// TIA Portal V16 export
// export: Created 2022-07-21T09:35:18.9169309Z, ExportSetting WithDefaults, DisplayName Totally Integrated Automation Portal, DisplayVersion V16 Update 4, DisplayName TIA Portal Version Control Interface, DisplayVersion V16 Update 2, DisplayName TIA Portal Openness, DisplayVersion V16 Update 4, DisplayName SINAMICS Startdrive Advanced, DisplayVersion V16 Update 5, DisplayName SINAMICS Startdrive G130, G150, S120, S150, SINAMICS MV, S210, DisplayVersion V16 Update 5, DisplayName SINAMICS Startdrive G110M, G120, G120C, G120D, G120P, G115D, DisplayVersion V16 Update 5, DisplayName STEP 7 Professional, DisplayVersion V16 Update 4, DisplayName STEP 7 Safety, DisplayVersion V16, DisplayName WinCC Advanced, DisplayVersion V16 Update 4
FUNCTION_BLOCK "fbVersaStandardCom"   // FB22, LAD
TITLE = Blok do komunikacji z Versa
{ S7_Optimized_Access := 'TRUE' }
VERSION : 0.1
// stored: AutoNumber true, IsIECCheckEnabled false, IsRetainMemResEnabled false, MemoryReserve 100, SetENOAutomatically false, UDAEnableTagReadback false
   VAR_INPUT
      hwAdr : HW_IO;   // Hardware ID modułu
      dataFromSafety : Bool;
      heaterOn : Bool;   // Załączenie grzałek (=1)
      motorsOn : Bool;   // Wszystkie silniki włącz (=1)
      pump1On : Bool;   // Udostępnienie silnika 1 ON (=1)
      pump2On : Bool;   // Udostępnienie silnika 2 ON (=1)
      standbyOn : Bool;   // Załącz czuwanie (=1)
      autoOn : Bool;   // Tryb automatyczny (=1)
      maxRpm : Int := 80;   // Maksymalna predkość pomp wg. nastaw Nordson
   END_VAR
   VAR_OUTPUT
      dataSendError : Bool;   // Bład podczas wysyłki TG
      dataReceiveError : Bool;   // Błąd podczas pobierania TG
      incorrectParam : Bool;   // Niepoprawne parametry do Nordsona
      SpeedLine1Perc : Int;   // Predkość linii po konwersji prędkości pompy
      SpeedLine2Perc : Int;   // Predkość linii po konwersji prędkości pompy
   END_VAR
   VAR_IN_OUT
      monitoringError : "typeNordsonMonitoring";
      device : "typeNordson";
   END_VAR
   VAR DB_SPECIFIC
      dataSend : "typeNordsonTGOut";
      dataReceive : "typeNordsonTGIn";
      hwAddress : HW_IO;
      retValRead : Int;
      retValSend : Int;
   END_VAR
   VAR_TEMP
      tpump1Speed : Int;   // Prędkość pompy 1
      tpump2Speed : Int;   // Prędkość pompy 2
      tFactor : Real;
      tpump1SpeedPerc : Int;   // Prędkość pompy 1
      tpump2SpeedPerc : Int;   // Prędkość pompy 2
      tMaxRpm : Real;
   END_VAR
   VAR_TEMP   // added for the SCL form of the ladder/FBD networks
      _w1 : Bool;
      _w2 : Bool;
   END_VAR
BEGIN

REGION Network 1: Załaduj adres modułu
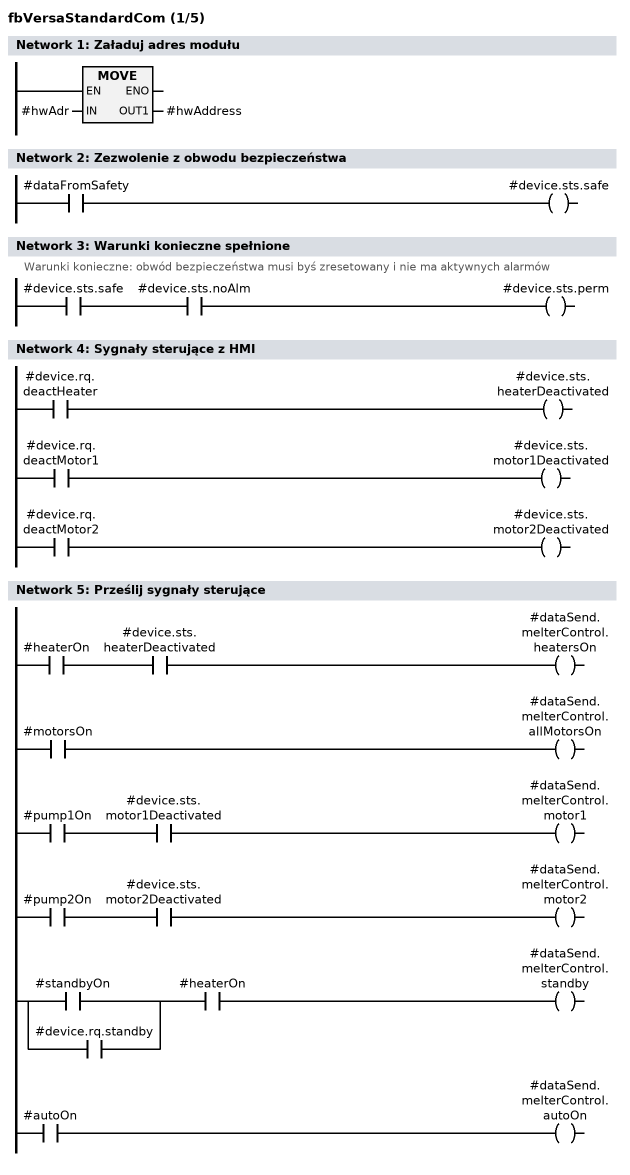
   RUNG wire#powerrail
      Move(in := #hwAdr, out1 => #hwAddress)
   END_RUNG
   // the same network as SCL:
   #hwAddress := #hwAdr;
END_REGION

REGION Network 2: Zezwolenie z obwodu bezpieczeństwa
   RUNG wire#powerrail
      Contact( #dataFromSafety )
      Coil( #device.sts.safe )
   END_RUNG
   // the same network as SCL:
   #device.sts.safe := #dataFromSafety;
END_REGION

REGION Network 3: Warunki konieczne spełnione
   // Warunki konieczne: obwód bezpieczeństwa musi byś zresetowany i nie ma aktywnych alarmów
   RUNG wire#powerrail
      Contact( #device.sts.safe )
      Contact( #device.sts.noAlm )
      Coil( #device.sts.perm )
   END_RUNG
   // the same network as SCL:
   #device.sts.perm := #device.sts.safe AND #device.sts.noAlm;
END_REGION

REGION Network 4: Sygnały sterujące z HMI
   RUNG wire#powerrail
      Contact( #device.rq.deactHeater )
      Coil( #device.sts.heaterDeactivated )
   END_RUNG
   RUNG wire#powerrail
      Contact( #device.rq.deactMotor1 )
      Coil( #device.sts.motor1Deactivated )
   END_RUNG
   RUNG wire#powerrail
      Contact( #device.rq.deactMotor2 )
      Coil( #device.sts.motor2Deactivated )
   END_RUNG
   // the same network as SCL:
   #device.sts.heaterDeactivated := #device.rq.deactHeater;
   #device.sts.motor1Deactivated := #device.rq.deactMotor1;
   #device.sts.motor2Deactivated := #device.rq.deactMotor2;
END_REGION

REGION Network 5: Prześlij sygnały sterujące
   RUNG wire#powerrail
      Contact( #heaterOn )
      Contact( #device.sts.heaterDeactivated )
      Coil( #dataSend.melterControl.heatersOn )
   END_RUNG
   RUNG wire#powerrail
      Contact( #motorsOn )
      Coil( #dataSend.melterControl.allMotorsOn )
   END_RUNG
   RUNG wire#powerrail
      Contact( #pump1On )
      Contact( #device.sts.motor1Deactivated )
      Coil( #dataSend.melterControl.motor1 )
   END_RUNG
   RUNG wire#powerrail
      Contact( #pump2On )
      Contact( #device.sts.motor2Deactivated )
      Coil( #dataSend.melterControl.motor2 )
   END_RUNG
   RUNG wire#powerrail
      Contact( #standbyOn )
      wire#w1
      Contact( #heaterOn )
      Coil( #dataSend.melterControl.standby )
   END_RUNG
   RUNG wire#powerrail
      Contact( #device.rq.standby )
   END_RUNG wire#w1
   RUNG wire#powerrail
      Contact( #autoOn )
      Coil( #dataSend.melterControl.autoOn )
   END_RUNG
   // the same network as SCL:
   #dataSend.melterControl.heatersOn := #heaterOn AND #device.sts.heaterDeactivated;
   #dataSend.melterControl.allMotorsOn := #motorsOn;
   #dataSend.melterControl.motor1 := #pump1On AND #device.sts.motor1Deactivated;
   #dataSend.melterControl.motor2 := #pump2On AND #device.sts.motor2Deactivated;
   #dataSend.melterControl.standby := (#standbyOn OR #device.rq.standby) AND #heaterOn;
   #dataSend.melterControl.autoOn := #autoOn;
END_REGION

REGION Network 6: Sprawdzanie maksymalnej prędkości 1
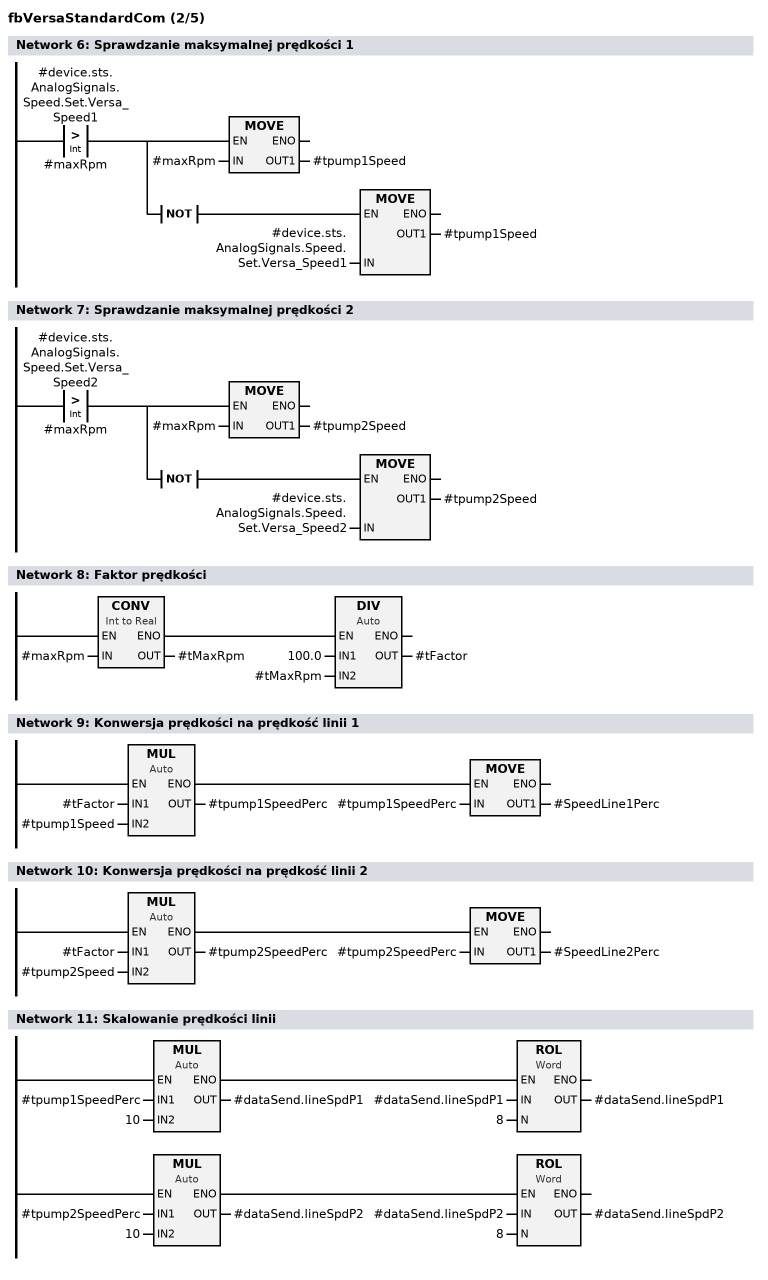
   RUNG wire#powerrail
      { S7_Templates := "SrcType := Int" } GT_Contact(in1 := #device.sts.AnalogSignals.Speed.Set.Versa_Speed1, in2 := #maxRpm)
      wire#w1
      Move(in := #maxRpm, out1 => #tpump1Speed)
   END_RUNG
   RUNG wire#w1
      Not()
      Move(in := #device.sts.AnalogSignals.Speed.Set.Versa_Speed1, out1 => #tpump1Speed)
   END_RUNG
   // the same network as SCL:
   #_w1 := #device.sts.AnalogSignals.Speed.Set.Versa_Speed1 > #maxRpm;
   IF #_w1 THEN #tpump1Speed := #maxRpm; END_IF;
   IF NOT #_w1 THEN #tpump1Speed := #device.sts.AnalogSignals.Speed.Set.Versa_Speed1; END_IF;
END_REGION

REGION Network 7: Sprawdzanie maksymalnej prędkości 2
   RUNG wire#powerrail
      { S7_Templates := "SrcType := Int" } GT_Contact(in1 := #device.sts.AnalogSignals.Speed.Set.Versa_Speed2, in2 := #maxRpm)
      wire#w1
      Move(in := #maxRpm, out1 => #tpump2Speed)
   END_RUNG
   RUNG wire#w1
      Not()
      Move(in := #device.sts.AnalogSignals.Speed.Set.Versa_Speed2, out1 => #tpump2Speed)
   END_RUNG
   // the same network as SCL:
   #_w1 := #device.sts.AnalogSignals.Speed.Set.Versa_Speed2 > #maxRpm;
   IF #_w1 THEN #tpump2Speed := #maxRpm; END_IF;
   IF NOT #_w1 THEN #tpump2Speed := #device.sts.AnalogSignals.Speed.Set.Versa_Speed2; END_IF;
END_REGION

REGION Network 8: Faktor prędkości
   RUNG wire#powerrail
      { S7_Templates := "[SrcType := Int, DestType := Real]" } Convert(in := #maxRpm, out => #tMaxRpm)
      Div(in1 := 100.0, in2 := #tMaxRpm, out => #tFactor)
   END_RUNG
   // the same network as SCL:
   #tMaxRpm := INT_TO_REAL(#maxRpm);
   #tFactor := 100.0 / #tMaxRpm;
END_REGION

REGION Network 9: Konwersja prędkości na prędkość linii 1
   RUNG wire#powerrail
      Mul(in1 := #tFactor, in2 := #tpump1Speed, out => #tpump1SpeedPerc)
      Move(in := #tpump1SpeedPerc, out1 => #SpeedLine1Perc)
   END_RUNG
   // the same network as SCL:
   #tpump1SpeedPerc := #tFactor * #tpump1Speed;
   #SpeedLine1Perc := #tpump1SpeedPerc;
END_REGION

REGION Network 10: Konwersja prędkości na prędkość linii 2
   RUNG wire#powerrail
      Mul(in1 := #tFactor, in2 := #tpump2Speed, out => #tpump2SpeedPerc)
      Move(in := #tpump2SpeedPerc, out1 => #SpeedLine2Perc)
   END_RUNG
   // the same network as SCL:
   #tpump2SpeedPerc := #tFactor * #tpump2Speed;
   #SpeedLine2Perc := #tpump2SpeedPerc;
END_REGION

REGION Network 11: Skalowanie prędkości linii
   #dataSend.lineSpdP1 := #tpump1SpeedPerc * 10;
   #dataSend.lineSpdP1 := ROL(IN := #dataSend.lineSpdP1, N := 8);
   #dataSend.lineSpdP2 := #tpump2SpeedPerc * 10;
   #dataSend.lineSpdP2 := ROL(IN := #dataSend.lineSpdP2, N := 8);
END_REGION

REGION Network 12: Wyślij dane
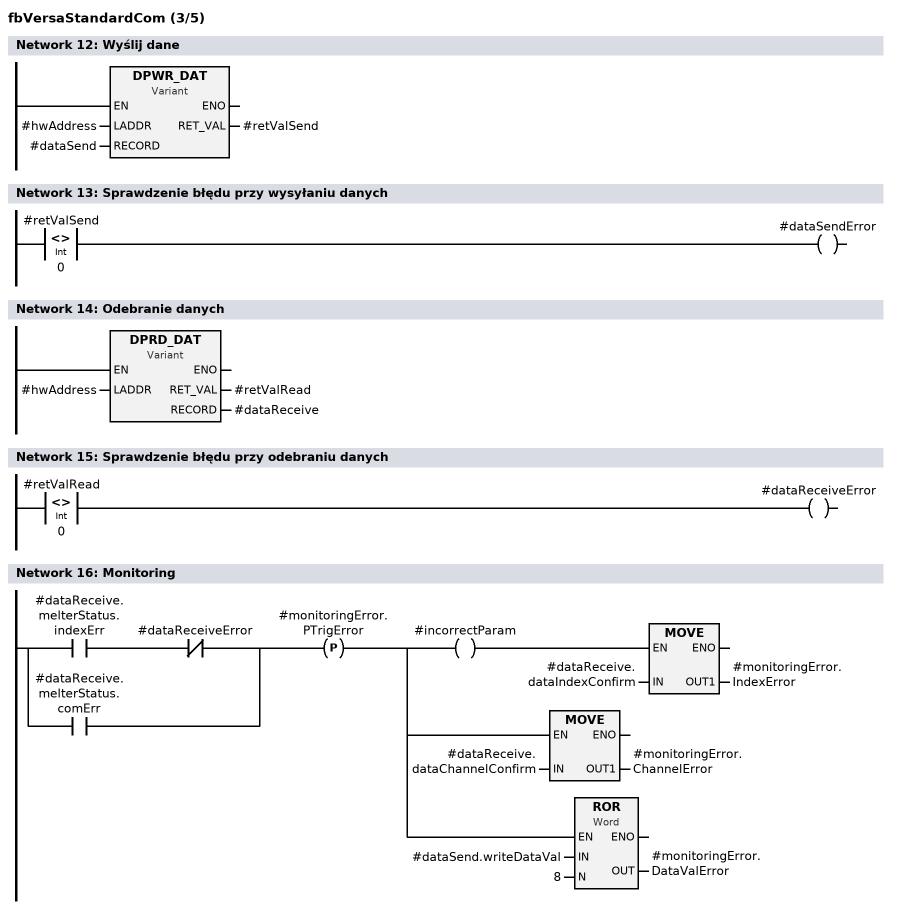
   RUNG wire#powerrail
      { S7_Templates := "[ptr_type := Variant, laddr_type := HW_IO]" } DPWR_DAT(LADDR := #hwAddress, RECORD := #dataSend, RET_VAL => #retValSend)
   END_RUNG
   // the same network as SCL:
   #retValSend := DPWR_DAT(LADDR := #hwAddress, RECORD := #dataSend);
END_REGION

REGION Network 13: Sprawdzenie błędu przy wysyłaniu danych
   RUNG wire#powerrail
      { S7_Templates := "SrcType := Int" } NE_Contact(in1 := #retValSend, in2 := 0)
      Coil( #dataSendError )
   END_RUNG
   // the same network as SCL:
   #dataSendError := #retValSend <> 0;
END_REGION

REGION Network 14: Odebranie danych
   RUNG wire#powerrail
      { S7_Templates := "[ptr_type := Variant, laddr_type := HW_IO]" } DPRD_DAT(LADDR := #hwAddress, RET_VAL => #retValRead, RECORD => #dataReceive)
   END_RUNG
   // the same network as SCL:
   #retValRead := DPRD_DAT(LADDR := #hwAddress, RECORD => #dataReceive);
END_REGION

REGION Network 15: Sprawdzenie błędu przy odebraniu danych
   RUNG wire#powerrail
      { S7_Templates := "SrcType := Int" } NE_Contact(in1 := #retValRead, in2 := 0)
      Coil( #dataReceiveError )
   END_RUNG
   // the same network as SCL:
   #dataReceiveError := #retValRead <> 0;
END_REGION

REGION Network 16: Monitoring
   #_w1 := (#dataReceive.melterStatus.indexErr AND NOT #dataReceiveError) OR #dataReceive.melterStatus.comErr;
   #_w2 := #_w1 AND NOT #monitoringError.PTrigError;   // rising edge
   #monitoringError.PTrigError := #_w1;
   #incorrectParam := #_w2;
   IF #_w2 THEN
       #monitoringError.IndexError := #dataReceive.dataIndexConfirm;
       #monitoringError.ChannelError := #dataReceive.dataChannelConfirm;
       #monitoringError.DataValError := ROR(IN := #dataSend.writeDataVal, N := 8);
   END_IF;
END_REGION

REGION Network 17: Statusy
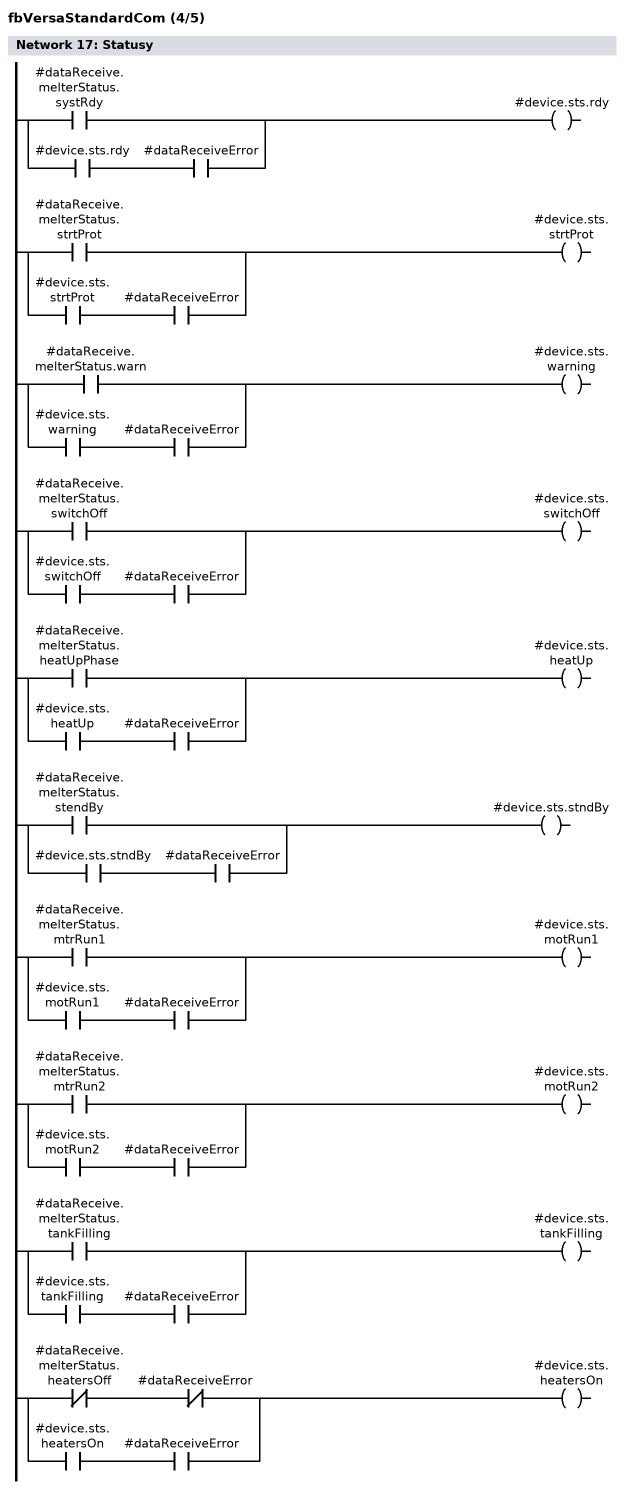
   RUNG wire#powerrail
      Contact( #dataReceive.melterStatus.systRdy )
      wire#w1
      Coil( #device.sts.rdy )
   END_RUNG
   RUNG wire#powerrail
      Contact( #device.sts.rdy )
      Contact( #dataReceiveError )
   END_RUNG wire#w1
   RUNG wire#powerrail
      Contact( #dataReceive.melterStatus.strtProt )
      wire#w2
      Coil( #device.sts.strtProt )
   END_RUNG
   RUNG wire#powerrail
      Contact( #device.sts.strtProt )
      Contact( #dataReceiveError )
   END_RUNG wire#w2
   RUNG wire#powerrail
      Contact( #dataReceive.melterStatus.warn )
      wire#w3
      Coil( #device.sts.warning )
   END_RUNG
   RUNG wire#powerrail
      Contact( #device.sts.warning )
      Contact( #dataReceiveError )
   END_RUNG wire#w3
   RUNG wire#powerrail
      Contact( #dataReceive.melterStatus.switchOff )
      wire#w4
      Coil( #device.sts.switchOff )
   END_RUNG
   RUNG wire#powerrail
      Contact( #device.sts.switchOff )
      Contact( #dataReceiveError )
   END_RUNG wire#w4
   RUNG wire#powerrail
      Contact( #dataReceive.melterStatus.heatUpPhase )
      wire#w5
      Coil( #device.sts.heatUp )
   END_RUNG
   RUNG wire#powerrail
      Contact( #device.sts.heatUp )
      Contact( #dataReceiveError )
   END_RUNG wire#w5
   RUNG wire#powerrail
      Contact( #dataReceive.melterStatus.stendBy )
      wire#w6
      Coil( #device.sts.stndBy )
   END_RUNG
   RUNG wire#powerrail
      Contact( #device.sts.stndBy )
      Contact( #dataReceiveError )
   END_RUNG wire#w6
   RUNG wire#powerrail
      Contact( #dataReceive.melterStatus.mtrRun1 )
      wire#w7
      Coil( #device.sts.motRun1 )
   END_RUNG
   RUNG wire#powerrail
      Contact( #device.sts.motRun1 )
      Contact( #dataReceiveError )
   END_RUNG wire#w7
   RUNG wire#powerrail
      Contact( #dataReceive.melterStatus.mtrRun2 )
      wire#w8
      Coil( #device.sts.motRun2 )
   END_RUNG
   RUNG wire#powerrail
      Contact( #device.sts.motRun2 )
      Contact( #dataReceiveError )
   END_RUNG wire#w8
   RUNG wire#powerrail
      Contact( #dataReceive.melterStatus.tankFilling )
      wire#w9
      Coil( #device.sts.tankFilling )
   END_RUNG
   RUNG wire#powerrail
      Contact( #device.sts.tankFilling )
      Contact( #dataReceiveError )
   END_RUNG wire#w9
   RUNG wire#powerrail
      I_Contact( #dataReceive.melterStatus.heatersOff )
      I_Contact( #dataReceiveError )
      wire#w10
      Coil( #device.sts.heatersOn )
   END_RUNG
   RUNG wire#powerrail
      Contact( #device.sts.heatersOn )
      Contact( #dataReceiveError )
   END_RUNG wire#w10
   // the same network as SCL:
   #device.sts.rdy := #dataReceive.melterStatus.systRdy OR (#device.sts.rdy AND #dataReceiveError);
   #device.sts.strtProt := #dataReceive.melterStatus.strtProt OR (#device.sts.strtProt AND #dataReceiveError);
   #device.sts.warning := #dataReceive.melterStatus.warn OR (#device.sts.warning AND #dataReceiveError);
   #device.sts.switchOff := #dataReceive.melterStatus.switchOff OR (#device.sts.switchOff AND #dataReceiveError);
   #device.sts.heatUp := #dataReceive.melterStatus.heatUpPhase OR (#device.sts.heatUp AND #dataReceiveError);
   #device.sts.stndBy := #dataReceive.melterStatus.stendBy OR (#device.sts.stndBy AND #dataReceiveError);
   #device.sts.motRun1 := #dataReceive.melterStatus.mtrRun1 OR (#device.sts.motRun1 AND #dataReceiveError);
   #device.sts.motRun2 := #dataReceive.melterStatus.mtrRun2 OR (#device.sts.motRun2 AND #dataReceiveError);
   #device.sts.tankFilling := #dataReceive.melterStatus.tankFilling OR (#device.sts.tankFilling AND #dataReceiveError);
   #device.sts.heatersOn := (NOT #dataReceive.melterStatus.heatersOff AND NOT #dataReceiveError) OR (#device.sts.heatersOn AND #dataReceiveError);
END_REGION

REGION Network 18: Aktywny system
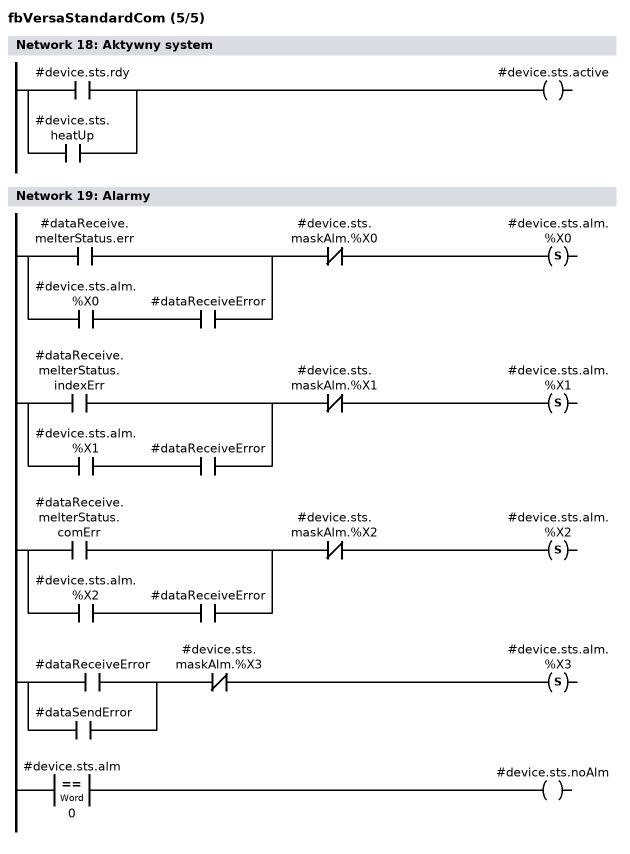
   RUNG wire#powerrail
      Contact( #device.sts.rdy )
      wire#w1
      Coil( #device.sts.active )
   END_RUNG
   RUNG wire#powerrail
      Contact( #device.sts.heatUp )
   END_RUNG wire#w1
   // the same network as SCL:
   #device.sts.active := #device.sts.rdy OR #device.sts.heatUp;
END_REGION

REGION Network 19: Alarmy
   RUNG wire#powerrail
      Contact( #dataReceive.melterStatus.err )
      wire#w1
      I_Contact( #device.sts.maskAlm.%X0 )
      S_Coil( #device.sts.alm.%X0 )
   END_RUNG
   RUNG wire#powerrail
      Contact( #device.sts.alm.%X0 )
      Contact( #dataReceiveError )
   END_RUNG wire#w1
   RUNG wire#powerrail
      Contact( #dataReceive.melterStatus.indexErr )
      wire#w2
      I_Contact( #device.sts.maskAlm.%X1 )
      S_Coil( #device.sts.alm.%X1 )
   END_RUNG
   RUNG wire#powerrail
      Contact( #device.sts.alm.%X1 )
      Contact( #dataReceiveError )
   END_RUNG wire#w2
   RUNG wire#powerrail
      Contact( #dataReceive.melterStatus.comErr )
      wire#w3
      I_Contact( #device.sts.maskAlm.%X2 )
      S_Coil( #device.sts.alm.%X2 )
   END_RUNG
   RUNG wire#powerrail
      Contact( #device.sts.alm.%X2 )
      Contact( #dataReceiveError )
   END_RUNG wire#w3
   RUNG wire#powerrail
      Contact( #dataReceiveError )
      wire#w4
      I_Contact( #device.sts.maskAlm.%X3 )
      S_Coil( #device.sts.alm.%X3 )
   END_RUNG
   RUNG wire#powerrail
      Contact( #dataSendError )
   END_RUNG wire#w4
   RUNG wire#powerrail
      { S7_Templates := "SrcType := Word" } EQ_Contact(in1 := #device.sts.alm, in2 := 0)
      Coil( #device.sts.noAlm )
   END_RUNG
   // the same network as SCL:
   IF (#dataReceive.melterStatus.err OR (#device.sts.alm.%X0 AND #dataReceiveError)) AND NOT #device.sts.maskAlm.%X0 THEN
       #device.sts.alm.%X0 := TRUE;
   END_IF;
   IF (#dataReceive.melterStatus.indexErr OR (#device.sts.alm.%X1 AND #dataReceiveError)) AND NOT #device.sts.maskAlm.%X1 THEN
       #device.sts.alm.%X1 := TRUE;
   END_IF;
   IF (#dataReceive.melterStatus.comErr OR (#device.sts.alm.%X2 AND #dataReceiveError)) AND NOT #device.sts.maskAlm.%X2 THEN
       #device.sts.alm.%X2 := TRUE;
   END_IF;
   IF (#dataReceiveError OR #dataSendError) AND NOT #device.sts.maskAlm.%X3 THEN
       #device.sts.alm.%X3 := TRUE;
   END_IF;
   #device.sts.noAlm := #device.sts.alm = 0;
END_REGION

REGION Network 20 (SCL): Alarmy dla temperatur

   //Czy wyświetlić alarm że temperatura jest powyzej/poniżej przyjętych limitów z poziomu HMI ?
   //Ruszt
   IF (#device.sts.AnalogSignals.Limits.Versa1_OL_Temp_Stemp < #device.sts.AnalogSignals.Temperature.Read.Versa_ActTemp_Stemp OR
       #device.sts.AnalogSignals.Limits.Versa1_UL_Temp_Stemp > #device.sts.AnalogSignals.Temperature.Read.Versa_ActTemp_Stemp) AND
       NOT #dataReceiveError AND NOT #device.sts.maskAlm.%X6 THEN

       #device.sts.alm.%X6 := TRUE;
   END_IF;

   //Pojemnik
   IF (#device.sts.AnalogSignals.Limits.Versa1_OL_Temp_Pump < #device.sts.AnalogSignals.Temperature.Read.Versa_ActTemp_Pump OR
       #device.sts.AnalogSignals.Limits.Versa1_UL_Temp_Pump > #device.sts.AnalogSignals.Temperature.Read.Versa_ActTemp_Pump) AND
       NOT #dataReceiveError AND NOT #device.sts.maskAlm.%X7 THEN

       #device.sts.alm.%X7 := TRUE;
   END_IF;

   //Wąż 1
   IF (#device.sts.AnalogSignals.Limits.Versa1_OL_Temp_Hose_1 < #device.sts.AnalogSignals.Temperature.Read.Versa_ActTemp_Hose_1 OR
       #device.sts.AnalogSignals.Limits.Versa1_UL_Temp_Hose_1 > #device.sts.AnalogSignals.Temperature.Read.Versa_ActTemp_Hose_1) AND
       NOT #dataReceiveError AND NOT #device.sts.maskAlm.%X8 THEN

       #device.sts.alm.%X8 := TRUE;
   END_IF;

   //Pistolet 1
   IF (#device.sts.AnalogSignals.Limits.Versa1_OL_Temp_HoseDistrib_1 < #device.sts.AnalogSignals.Temperature.Read.Versa_ActTemp_HoseDistrib_1 OR
       #device.sts.AnalogSignals.Limits.Versa1_UL_Temp_HoseDistrib_1 > #device.sts.AnalogSignals.Temperature.Read.Versa_ActTemp_HoseDistrib_1) AND
       NOT #dataReceiveError AND NOT #device.sts.maskAlm.%X9 THEN

       #device.sts.alm.%X9 := TRUE;
   END_IF;

   //Wąż 2
   IF (#device.sts.AnalogSignals.Limits.Versa1_OL_Temp_Hose_2 < #device.sts.AnalogSignals.Temperature.Read.Versa_ActTemp_Hose_2 OR
       #device.sts.AnalogSignals.Limits.Versa1_UL_Temp_Hose_2 > #device.sts.AnalogSignals.Temperature.Read.Versa_ActTemp_Hose_2) AND
       NOT #dataReceiveError AND NOT #device.sts.maskAlm.%X10 THEN

       #device.sts.alm.%X10 := TRUE;
   END_IF;

   //Pistolet 2
   IF (#device.sts.AnalogSignals.Limits.Versa1_OL_Temp_HoseDistrib_2 < #device.sts.AnalogSignals.Temperature.Read.Versa_ActTemp_HoseDistrib_2 OR
       #device.sts.AnalogSignals.Limits.Versa1_UL_Temp_HoseDistrib_2 > #device.sts.AnalogSignals.Temperature.Read.Versa_ActTemp_HoseDistrib_2) AND
       NOT #dataReceiveError AND NOT #device.sts.maskAlm.%X11 THEN

       #device.sts.alm.%X11 := TRUE;
   END_IF;

   //Wąż 3
   IF (#device.sts.AnalogSignals.Limits.Versa1_OL_Temp_Zone7 < #device.sts.AnalogSignals.Temperature.Read.Versa_ActTemp_Zone7 OR
       #device.sts.AnalogSignals.Limits.Versa1_UL_Temp_Zone7 > #device.sts.AnalogSignals.Temperature.Read.Versa_ActTemp_Zone7) AND
       NOT #dataReceiveError AND NOT #device.sts.maskAlm.%X12 THEN

       #device.sts.alm.%X12 := TRUE;
   END_IF;

   //Pistolet 3
   IF (#device.sts.AnalogSignals.Limits.Versa1_OL_Temp_Zone8 < #device.sts.AnalogSignals.Temperature.Read.Versa_ActTemp_Zone8 OR
       #device.sts.AnalogSignals.Limits.Versa1_UL_Temp_Zone8 > #device.sts.AnalogSignals.Temperature.Read.Versa_ActTemp_Zone8) AND
       NOT #dataReceiveError AND NOT #device.sts.maskAlm.%X13 THEN

       #device.sts.alm.%X13 := TRUE;
   END_IF;

   //Wąż 4
   IF (#device.sts.AnalogSignals.Limits.Versa1_OL_Temp_Zone9 < #device.sts.AnalogSignals.Temperature.Read.Versa_ActTemp_Zone9 OR
       #device.sts.AnalogSignals.Limits.Versa1_UL_Temp_Zone9 > #device.sts.AnalogSignals.Temperature.Read.Versa_ActTemp_Zone9) AND
       NOT #dataReceiveError AND NOT #device.sts.maskAlm.%X14 THEN

       #device.sts.alm.%X14 := TRUE;
   END_IF;

   //Pistolet 4
   IF (#device.sts.AnalogSignals.Limits.Versa1_OL_Temp_Zone10 < #device.sts.AnalogSignals.Temperature.Read.Versa_ActTemp_Zone10 OR
       #device.sts.AnalogSignals.Limits.Versa1_UL_Temp_Zone10 > #device.sts.AnalogSignals.Temperature.Read.Versa_ActTemp_Zone10) AND
       NOT #dataReceiveError AND NOT #device.sts.maskAlm.%X15 THEN

       #device.sts.alm.%X15 := TRUE;
   END_IF;
END_REGION

REGION Network 21 (SCL): Reset alarmów
   #device.sts.alm := #device.sts.alm AND NOT #device.rq.almAck;
END_REGION
END_FUNCTION_BLOCK
